(* PLC project codesysParallelTest.project, CODESYS CODESYS V3.5 SP17 Patch 3 *)
(* stored: creationDateTime 2022-12-13T23:13:44.5126035, modificationDateTime 2022-12-11T22:42:34.2824338 *)

PROGRAM flow_11

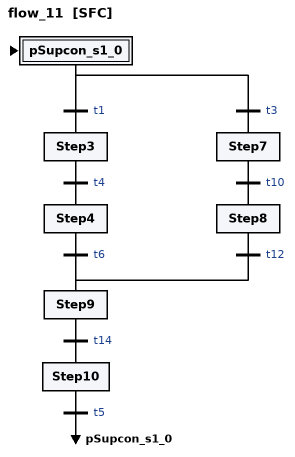
INITIAL_STEP pSupcon_s1_0:
END_STEP
TRANSITION FROM pSupcon_s1_0 TO Step3
  := t1;
END_TRANSITION
TRANSITION FROM pSupcon_s1_0 TO Step7
  := t3;
END_TRANSITION
STEP Step3:
END_STEP
TRANSITION FROM Step3 TO Step4
  := t4;
END_TRANSITION
STEP Step4:
END_STEP
TRANSITION FROM Step4 TO Step9
  := t6;
END_TRANSITION
STEP Step7:
END_STEP
TRANSITION FROM Step7 TO Step8
  := t10;
END_TRANSITION
STEP Step8:
END_STEP
TRANSITION FROM Step8 TO Step9
  := t12;
END_TRANSITION
STEP Step9:
END_STEP
TRANSITION FROM Step9 TO Step10
  := t14;
END_TRANSITION
STEP Step10:
END_STEP
TRANSITION FROM Step10 TO pSupcon_s1_0
  := t5;
END_TRANSITION
END_PROGRAM
